// TIA Portal V20 export
TYPE "type_emRelations_em2_cmStatus"
// stored: Access Published, Namespace Unit1
   STRUCT
      JROutPnPLeftSafetyPin : "LBC_typeDigitalSignalControlNode";
      JROutPnPLeftJRDetect : "LBC_typeDigitalSignalControlNode";
      JROutPnPRightSafetyPin : "LBC_typeDigitalSignalControlNode";
      JROutPnPRightJRDetect : "LBC_typeDigitalSignalControlNode";
      JROutPnPLeftAxisX : "LBC_typeAxis64PosControlNode";
      JROutPnPLeftAxisZ : "LBC_typeAxis64PosControlNode";
      JROutPnPRightAxisX : "LBC_typeAxis64PosControlNode";
      JROutPnPRightAxisZ : "LBC_typeAxis64PosControlNode";
      JROutPnPLeftClampOpenClose : "LBC_typeTwoWayActuatorControlNode";
      JROutPnPRightClampOpenClose : "LBC_typeTwoWayActuatorControlNode";
      PowerMeter : "LER_typePAC3220ControlNode";
   END_STRUCT;
END_TYPE
